Universal Robots URScript: test.script

def unnamed():
  global _hidden_verificationVariable=0
  set_safety_mode_transition_hardness(1)
  set_target_payload(0.100000, [0.000000, 0.000000, 0.000000], [0.000033, 0.000033, 0.000033, 0.000000, 0.000000, 0.000000])
  set_tool_communication(False, 115200, 0, 1, 1.5, 3.5)
  set_tool_output_mode(0)
  set_tool_digital_output_mode(0, 1)
  set_tool_digital_output_mode(1, 1)
  set_tool_voltage(0)
  modbus_add_signal("192.168.1.101", 255, 0, 2, "MODBUS_1", False)
  modbus_set_signal_update_frequency("MODBUS_1", 10)
  modbus_add_signal("192.168.1.101", 255, 0, 2, "MODBUS_2", False)
  modbus_set_signal_update_frequency("MODBUS_2", 10)
  set_gravity([0.0, 0.0, 9.82])
  set_tcp(p[0.0,0.0,0.0,0.0,0.0,0.0])
  set_standard_analog_input_domain(0, 1)
  set_standard_analog_input_domain(1, 1)
  set_tool_analog_input_domain(0, 1)
  set_tool_analog_input_domain(1, 1)
  set_analog_outputdomain(0, 0)
  set_analog_outputdomain(1, 0)
  set_input_actions_to_default()
  global tschauhome=p[0.09193868628606418,-0.13209828878395144,0.693632573899399,-1.2079453233871906,1.2128578750035333,-1.2059658490999983]
  step_count_f147a8f9_8b71_40fa_91a0_298106da69ef = 0.0
  thread Step_Counter_Thread_a6a4bf7a_6eaa_46fd_8e32_1aaa87d76119():
    while (True):
      step_count_f147a8f9_8b71_40fa_91a0_298106da69ef = step_count_f147a8f9_8b71_40fa_91a0_298106da69ef + 1.0
      sync()
    end
  end
  run Step_Counter_Thread_a6a4bf7a_6eaa_46fd_8e32_1aaa87d76119()
  global Waypoint_1_p=p[-.288777179692, -.179779966064, .582810229051, -1.019466805800, -1.305578187210, .900389041639]
  global Waypoint_1_q=[0.2527463734149933, -1.3508151781610032, 0.8132980505572718, -2.5939046345152796, -1.9068782965289515, -0.3196676413165491]
  global Waypoint_2_p=p[-.413039328074, -.215094695379, .363792480527, -1.037272342104, -1.227684892797, 1.097662848233]
  global Waypoint_2_q=[0.24483251571655273, -0.8276537221721192, 1.1059377829181116, -3.492258688012594, -1.8283394018756312, -0.19470292726625615]

  $ 1 "Robot Program"
  $ 2 "MoveJ"
  $ 3 "Waypoint_1" "breakAfter"
  movej(get_inverse_kin(Waypoint_1_p, qnear=Waypoint_1_q), a=1.3962634015954636, v=1.0471975511965976)
  $ 4 "Waypoint_2" "breakAfter"
  movej(get_inverse_kin(Waypoint_2_p, qnear=Waypoint_2_q), a=1.3962634015954636, v=1.0471975511965976)
end
